//****************************************************************************************************
// Code generated by SFC Generator V1.13 on 02/04/18 16:19:18 by  MAC_IZZ from File D:\Rieckermann\old\Visio SFC\Snippet_Code\SEQ_HDR.txt
//****************************************************************************************************
//****************************************************************************************************

//================================ SEQ HEADER ================================//
//            Copyright 2018 Rieckermann Engineering Operations               //
//----------------------------------------------------------------------------//
// Title: UO_SIP_MX                                                       //
//                                                                            //
// Description:                                                               //
// Parent synchronisation flag indicating path set for filling line CIP                                                        //
//                                                                            //
// // SFC Revision History:
// Rev By               Date        CC         Note
// 0.1 Gerald Kontriner 07-Sep-2009            SFC structural design                                                       //
//----------------------------------------------------------------------------//
// Sequencer Revision History:                                                //
// Rev By               Date        CC        Note                            //
// 2.0 David Paspa      05-Jan-2018 NA        Reboot for S7-1500.             //
// 1.6 Khairul Basar    19-Nov-2009 NA        Reset #sqSequencer.STEP.Active  //
//                                            when STEP Finished.             //
// 1.5 Khairul Basar    15-Oct-2009 NA        Placeholder inserted:           //
//                                            "udtSQ_UO";          //
// 1.4 Khairul Basar    06-Oct-2009 NA        R #PAUSE;                       //
// 1.3 Khairul Basar    30-Sep-2009 NA        SEQ_HDR change STEP-0 code      //
//                                            deleted.                        //
// 1.2 Khairul Basar    26-Sep-2009 NA        Refer R4.                       //
// 1.1 Khairul Basar    23-Sep-2009 NA        Refer R3.                       //
// 1.0 Khairul Basar    20-Sep-2009 NA        STEP.Finished flag reset by     //
//                                            JUMP_MAN.                       //
// 0.9 Khairul Basar    11-Sep-2009 NA        SQ_TIMER added as VAR, declared //
//                                            in SEQ_FTR.                     //
// 0.8 Khairul Basar    09-Sep-2009 NA        SqSequencer.Err_Fault is reset  //
//                                            on Stop cmd, Step-0 dead code   //
//                                            deleted from ACT & Verify.      //
//                                            STP_FTR Step_withErr flag       //
//                                            STEP_NUM place holder           //
//                                            configured.                     //
// 0.7 Khairul Basar    28-Aug-2009 NA        SQ_FINISHED OUT added again.    //
//                                            Deleted during major mod R3.    //
// 0.6 Khairul Basar    23-Aug-2009 NA        Refer R2.                       //
// 0.5 Khairul Basar    23-Aug-2009 NA        Refer R1.                       //
// 0.4 Khairul Basar    18-Aug-2009 NA        Reset Step done with/out error  //
//                                            bits using FC:RSET.             //
// 0.3 David Paspa      16-Aug-2009 NA        Added placeholders for header   //
//                                            name and version and revision   //
//                                            history.                        //
// 0.2 Khairul Basar    11-Aug-2009 NA        Retired external udt file for   //
//                                            Static type parameters. All     //
//                                            parameters now IN, OUT or       //
//                                            IN_OUT.                         //
// 0.1 Khairul Basar    12-Jun-2009 NA        Initial design.                 //
//----------------------------------------------------------------------------//
// R4:                                                                        //
// 1.If SQ not finished Resume command will start Step timer, and redo the    //
// last action, verify the feedback.                                          //
// 2."STEP.finished" flag is ANDed with "TRN_AND_JUMP" in the snippet file    //
// TRN_HDR.This is to avoid checking of transition logic if STEP is not       //
// finished yet.                                                              //
// 3.MDCH, Load & transfer typo corrected.                                    //
//                                                                            //
// R3:                                                                        //
// 1.SqStepTimer.IN is reset in STEP_FTR instead of resetting it in TRN_HDR.  //
// This is because TRN_HDTR is not included in the Last step and StepTimer    //
// must reset in the last step.                                               //
// 2.Reset all the timers when SQ stops.Reset done in SEQ_HDR.                //
// Also STEP-finished flag reset when SQ is OFF to                            //
// scan last step.                                                            //
//                                                                            //
// R2:                                                                        //
// 1.Any step error will send the Sequencer into Pause state.Code added in    //
// SEQ_HDR.Snippet Place holder for Bool-array 8 is   //
// deleted.                                                                   //
//                                                                            //
// R1:                                                                        //
// 1.sqStepTimer:All Verification Code must satisfy the condition finish step //
// action within STEP_DELAY time(40s).If step actions not finished within the //
// time period the error flag will raise High signal.Else timer will reset.   //
// 2.sqRunTimer Added therefore can be used as retentive & non retentive.     //
// 3.sqSequencer: This is re-structured UDT which is redefined the symbol     //
// names as well as it gives more clearity.                                   //
// 4.fcMODE and fcCMD functions are added to handle the mode & command        //
// independently regardless of other logic.Two separate UDT udtMODE & udt     //
// CMD assigned to Mode & command function respectively.                      //
// 5.MAN_JUMP programed for manual mode jump operation with or without        //
// Transition code satisfied.TRN_AND_JUMP & NO_VERIFC are the parameters      //
// which will define whether verification code & transition code need to be   //
// checked to perform jump operation.                                         //
// 6.Auto to Manual switchover will be bumpless & will not affect step        //
// operation.Manual to auto switchover can be used to resume Step action at   //
// defined.                                                                   //
// Step number entered in STEPNO_JUMP.                                        //
//                                                                            //
// Parameters:                                                                //
// INPUTS                                                                     //
// ======                                                                     //
// SQ_CMD          Sequence command input inherited from object block         //
//                 0: off/idle                                                //
//                 1: start/initiate                                          //
//                 2: pause                                                   //
//                 3: resume                                                  //
//                 4: reserved (not programmed)                               //
//                 5: reserved (not programmed)                               //
//                 6: abort/go to last step                                   //
//                 7: acknowledge error/fault                                 //
// SQ_MODE         Sequencer Auto/Manual input inherited from object block    //
//                 1: manual                                                  //
//                 2: auto                                                    //
//                                                                            //
// INPUT/OUTPUTS                                                              //
// =============                                                              //
// SQ_JUMP_MAN     Allows manual jumping from one step to the next step. The  //
//                 manual jump flag is ORed with the transition process       //
//                 condition and so can be used to bypass the condition if the//
//                 sequence will not progress.                                //
//                 This input can also be used to jump to any step even       //
//                 when no transition -> step linkage exists. This is only    //
//                 possible when the SQ_MODE is in manual and SQ is in the    //
//                 idle step. The step to jump to is specified in             //
//                 SQ_man_jump_to_step (not accesseble by this FB in/out      //
//                 interface but a separate DB memory location).              //
//                                                                            //
// OUTPUTS                                                                    //
// =======                                                                    //
// SQ_STATE        The calculated state of the sequence                       //
//                 0: off/idle                                                //
//                 1: start/initiated                                         //
//                 2: paused                                                  //
//                 3: resumed                                                 //
//                 4: reserved (wrong Mode)                                   //
//                 5: reserved (Wrong commad)                                 //
//                 6: aborted/go to last step                                 //
//                 7: acknowledged error/fault                                //
// CURSTEP         Current step being proccessed.                             //
// S_ACTIVE        If current step is active                                  //
// NXT_STEP        Next step to jump to if transition condition is true       //
// ERR_FAULT       True if any error/ or fault present                        //
// PAUSED          True if step is paused                                     //
// OFF_IDLE        Sequence is not running but ready for next SQ (in step=0)  //
//----------------------------------------------------------------------------//
// Define variables:                                                          //
//----------------------------------------------------------------------------//
FUNCTION_BLOCK "fbUO_MFL_SIP_MX"
TITLE = UO : MFL_SIP_MX
NAME : FUSMX
AUTHOR : REO
VERSION : 0.1

VAR_INPUT
  MODE : INT :=2;
  SQ_CMD : INT :=0;
    _SIP_timer_complete_mx :BOOL ;	//Description
    _AUX_COND_EXn007_CMD :BOOL ;	//Description
    _TIME_DRAIN_PULSE :TIME ;	//Drain Time Setpoint
    _steam_compl_MFL_Mx :BOOL ;	//Parent synchronisation flag indicating SIP steaming is complete
    _pulse_drain_MFL_Mx :BOOL ;	//Flag indicating drain valve should be pulsed
    _ready_sip_MFL_Mx :BOOL ;	//Parent synchronisation flag for ready to start SIP
    _DEV_STATE_EXn007 :INT ;	//Device State of EXn007

END_VAR
VAR_OUTPUT
  SQ_STATE : INT ;
  CURSTEP : INT ;
  NXT_STEP : INT ;
  S_ACTIVE : BOOL ;
  ERR_FAULT : BOOL ;
  PAUSED : BOOL ;
  OFF_IDLE : BOOL ;
  SQ_FINISHED : BOOL ;
    _AUX_COND_EXn007 :BOOL ;	//Description
    _pulse_dr_compl_MFL_Mx :BOOL ;	//Pulsing of drain valve is complete
    _ready_steam_trap_MFL_Mx :BOOL ;	//Flag indicating steam traps are open
    _CMD_EXn007 :INT ;	//Command to EXn007
    _SUB_EXn007 :INT ;	//Substate selection to EXn007

END_VAR
VAR_IN_OUT
  STEPNO_JUMP : INT ;
  MAN_JUMP : BOOL ;
  NO_VERIFIC : BOOL ;
  TRN_AND_JUMP : BOOL ;

END_VAR
VAR
  sqStepTimer : "TON";
  sqRunTimer : "fbRunTimer";
  sqSequencer : "udtSQ_UO";
  SQ_TIMER: "TON";

END_VAR
BEGIN
NETWORK
TITLE =Call Mode checking function
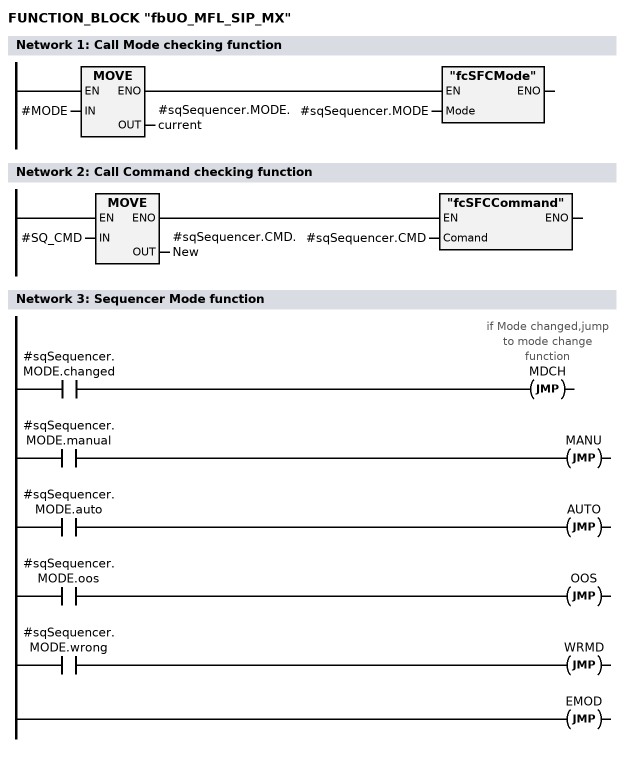

      L     #MODE;
      T     #sqSequencer.MODE.current;
      CALL "fcSFCMode" (
           Mode                     := #sqSequencer.MODE);

NETWORK
TITLE =Call Command checking function

      L     #SQ_CMD;
      T     #sqSequencer.CMD.New;

      CALL "fcSFCCommand" (
           Comand                   := #sqSequencer.CMD);

NETWORK
TITLE =Sequencer Mode function

      A     #sqSequencer.MODE.changed;
      JC    MDCH; // if Mode changed,jump to mode change function
      A     #sqSequencer.MODE.manual;
      JC    MANU;
      A     #sqSequencer.MODE.auto;
      JC    AUTO;
      A     #sqSequencer.MODE.oos;
      JC    OOS;
      A     #sqSequencer.MODE.wrong;
      JC    WRMD;
      JU    EMOD;

NETWORK
//----------------------------------------------------------------------------//
// On positive edge of mode change , this will execute once, only one cycle   //
// before going to execute the selected mode function below:                  //
//----------------------------------------------------------------------------//
TITLE =Mode change function
MDCH: NOP   0;
      SET   ;
      R     #sqStepTimer.IN;
      L     #sqSequencer.STEP.NumberCurrent;
      T     #STEPNO_JUMP;
      JU    EMOD;

NETWORK
//----------------------------------------------------------------------------//
// #TRN_AND_JUMP=can set/reset                                                //
// #sqSequencer.STEP.JumpCtrl=Can set/reset by #MAN_JUMP                      //
// #NO_VERIFIC=Can set/ Reset                                                 //
//----------------------------------------------------------------------------//
TITLE =Manual Mode function
MANU: NOP   0; //Manual mode selected



      A     #MAN_JUMP;
      =     #sqSequencer.STEP.JumpCtrl;
      A     #MAN_JUMP;
      JCN   EMOD;

      L     #STEPNO_JUMP;
      T     #sqSequencer.STEP.NumberNext;
      T     #sqSequencer.STEP.NumberCurrent;
      R     #MAN_JUMP; //Reset MAN_JUMP after loading user destination Step number
      R     #sqSequencer.STEP.Finished; //Reset finish flag, to execute next step action
      JU    EMOD;

NETWORK
//----------------------------------------------------------------------------//
// #TRN_AND_JUMP=always set                                                   //
// #sqSequencer.STEP.JumpCtrl=Always set                                      //
// #NO_VERIFIC=Alwasy Reset                                                   //
//----------------------------------------------------------------------------//
TITLE =Auto Mode function
AUTO: NOP   0; //Auto mode selected



      R     #MAN_JUMP;
      S     #TRN_AND_JUMP;
      R     #NO_VERIFIC;
      S     #sqSequencer.STEP.JumpCtrl; //Always Set in auto mode

      L     #sqSequencer.STEP.NumberCurrent;
      T     #STEPNO_JUMP;
      JU    EMOD;
NETWORK
TITLE =OOS mode function

OOS:  NOP   0; // Out of service
      JU    EMOD;
WRMD: NOP   0; //Wrong mode selected
      S     #sqSequencer.Error_Fault;
      L     "dbCONST_VAL".SQ_STATE.WRMODE;
      T     #SQ_STATE;

      JU    EMOD;

NETWORK
TITLE =Mode not changedd

      NOP   0;

NETWORK
TITLE =End Mode function

EMOD: NOP   0;

NETWORK
TITLE =An error will Pause the Sequencer,Operator must Resume SQ to run

      A     #sqSequencer.Error_Fault;
      AN    #sqSequencer.CMD.Changed;
      JC    PAUS;

NETWORK
TITLE =Command Action function

      A     #sqSequencer.CMD.Changed;
      JCN   CNCH; // if Command not changed,jump to end function
      R     #sqStepTimer.IN;


      A     #sqSequencer.CMD.Start;
      JC    STRT;

      A     #sqSequencer.CMD.Stop;
      JC    STOP;


      A     #sqSequencer.CMD.Pause;
      JC    PAUS;

      A     #sqSequencer.CMD.Resume;
      JC    RESM;

      A     #sqSequencer.CMD.Abort;
      JC    ABRT;

      A     #sqSequencer.CMD.Ack;
      JC    ACKN;

      A     #sqSequencer.CMD.wrong;
      JC    WCMD;

      JU    ECMD; //Wrong command/not specified command
//End Comand function

NETWORK
TITLE =Comand -Start/Initiate action function

STRT: NOP   0;
      R     #OFF_IDLE;
      R     #PAUSED;
      R     #sqSequencer.STEP.Active;
      R     #sqSequencer.STEP.Finished;
      R     #sqSequencer.STEP.ActionFinished;
      R     #sqSequencer.STEP.Jump;
      R     #sqSequencer.STEP.TimerExpired;
      R     #sqSequencer.STEP.Error_Fault;
      R     #sqSequencer.STEP.ActionVerified;
      R     #sqStepTimer.IN;

      S     #sqRunTimer.RESET;

//----------------------------------------------------------------------------//
// Load Initial step Number:                                                  //
//----------------------------------------------------------------------------//
      L     1;
      T     #sqSequencer.STEP.Initial;
      L     #sqSequencer.STEP.Initial;
      T     #sqSequencer.STEP.NumberCurrent;
      T     #sqSequencer.STEP.NumberNext;




      L     "dbCONST_VAL".SQ_STATE.STARTED;
      T     #SQ_STATE;

//----------------------------------------------------------------------------//
// Reset Step done without error bits:                                        //
//----------------------------------------------------------------------------//
      CALL "RSET" (
           S_BIT                    := #sqSequencer.STEP.Done[1],
           N                        := 3);//Upto final step


//----------------------------------------------------------------------------//
// Reset Step done with error bits:                                           //
//----------------------------------------------------------------------------//
      CALL "RSET" (
           S_BIT                    := #sqSequencer.STEP.WithError[1],
           N                        := 3);//Upto final step

      JU    ECMD; //End Function

NETWORK
TITLE =Comand -Stop action function

STOP: NOP   0;
      S     #OFF_IDLE;
      R     #sqSequencer.STEP.Active;
      R     #sqSequencer.STEP.Finished;
      R     #sqSequencer.STEP.ActionFinished;
      R     #sqSequencer.STEP.Jump;
      R     #sqSequencer.STEP.TimerExpired;
      R     #sqSequencer.STEP.Error_Fault;
      R     #sqSequencer.Error_Fault;
      R     #sqSequencer.STEP.ActionVerified;
      R     #sqRunTimer.ENABLE;
      R     #sqStepTimer.IN;
      R     #SQ_TIMER.IN;
      R     #PAUSED;


//Go to last step
      L     3;
      T     #sqSequencer.FinalStep;
      L     #sqSequencer.FinalStep;
      T     #sqSequencer.STEP.NumberNext;
      L     "dbCONST_VAL".SQ_STATE.OFF_IDLE;
      T     #SQ_STATE;

      JU    ECMD; //End Function

NETWORK
TITLE =Comand -Pause action function

PAUS: NOP   0;
      S     #PAUSED;
      R     #S_ACTIVE;
      S     #sqRunTimer.PAUSE;
      L     #sqSequencer.STEP.NumberCurrent;
      T     #STEPNO_JUMP;
      L     "dbCONST_VAL".SQ_STATE.PAUSED;
      T     #SQ_STATE;

      JU    ECMD; //End Function

NETWORK
TITLE =Comand -Resume action function

RESM: NOP   0;
      R     #PAUSED;
      R     #sqRunTimer.PAUSE;
      R     #sqStepTimer.IN; //Reset Step timer
      L     "dbCONST_VAL".SQ_STATE.RESUMED;
      T     #SQ_STATE;

      A     #SQ_FINISHED;
      JC    ECMD;
      R     #sqSequencer.STEP.Active;
      R     #sqSequencer.STEP.Finished;
      R     #sqSequencer.STEP.ActionFinished;

      JU    ECMD; //End Function

NETWORK
TITLE =Comand -Abort action function

ABRT: NOP   0;
      L     "dbCONST_VAL".SQ_STATE.ABORTED;
      T     #SQ_STATE;

      JC    STOP; //Stop & Abort same
      JU    ECMD;

NETWORK
TITLE =Comand -Acknowledge action function

ACKN: NOP   0;
      R     #ERR_FAULT;
      R     #sqSequencer.Error_Fault;
      L     "dbCONST_VAL".SQ_STATE.ACKNOWLEDGED;
      T     #SQ_STATE;

      JU    ECMD; //End Function

NETWORK
TITLE =Comand -wrong/unavailable

WCMD: NOP   0;

      S     #sqSequencer.Error_Fault;
      L     "dbCONST_VAL".SQ_STATE.WRCMD;
      T     #SQ_STATE;

      JU    ECMD;
NETWORK
TITLE =Comand -not changedd

CNCH: NOP   0; // Command not changed

NETWORK
TITLE =End command Function

ECMD: NOP   0;

NETWORK
//----------------------------------------------------------------------------//
// Sequencer step jump list. Load the step number to execute the step:        //
//----------------------------------------------------------------------------//
TITLE =Sequencer Step Jump distrubution list
      L     #sqSequencer.STEP.NumberCurrent;
      JL    SQER; // If Sequencer Step number invalid or greater than available number of step
      JU    S000; // Exceptional Error Handling
      JU    S001; // STEP-001:
JU    S002; // STEP-002:
JU    S003; // STEP-003:


//----------------------------------------------------------------------------//
// If Step number is Invalid or Out of Range:                                 //
//----------------------------------------------------------------------------//
SQER: NOP   0;
      S     #sqSequencer.Error_Fault;
      JU    COMM; // Jump to Common Sequencer code handling function

NETWORK
//----------------------------------------------------------------------------//
// STEP0 STEP0 STEP0 STEP0 STEP0 STEP0 STEP0 STEP0 STEP0 STEP0 STEP0 STEP0 ST //
// STEP0 STEP0 STEP0 STEP0 STEP0 STEP0 STEP0 STEP0 STEP0 STEP0 STEP0 STEP0 ST //
// STEP0 STEP0 STEP0 STEP0 STEP0 STEP0 STEP0 STEP0 STEP0 STEP0 STEP0 STEP0 ST //
//----------------------------------------------------------------------------//
TITLE =STEP0 STEP0 STEP0 STEP0 STEP0 STEP0 STEP0 STEP0 STEP0 STEP0 STEP

NETWORK
TITLE =S000: STEP0::If Paused exit

S000: NOP   0;

      JU    COMM;






NETWORK
//================================ STEP HEADER ===============================//
// STEP001 STEP001 STEP001 STEP001 ST //
// STEP001 STEP001 STEP001 STEP001 ST //
// STEP001 STEP001 STEP001 STEP001 ST //
//----------------------------------------------------------------------------//
// Set EXx014 to substate FILTER.
Set ETx003 to State DRAIN.
Open Valve DVx173.

Flag parent ready to start SIP by setting synchronization flag SIP_ready.
//----------------------------------------------------------------------------//
TITLE =S001: STEP-01::MMFLx_UO_SIP: SIP of MMFLx commenced

S001: NOP   0;

      A     #sqSequencer.CMD.Pause; //If paused jump
      JC    COMM;

NETWORK
TITLE =S001:STEP-01:Begin Action

      A     #sqSequencer.STEP.Finished;
      JC    A001; // Exit Action code, Jump to A001 Transition code

      //----------------------------------------------------------------------//
      // Begin step Action:                                                   //
      //----------------------------------------------------------------------//
      A     #sqSequencer.STEP.Active;
      JC    L001; // Action number loaded, Jump to L001--Step Action List

      //----------------------------------------------------------------------//
      // Load Default/Initial Step action number:                             //
      //----------------------------------------------------------------------//
      S     #sqSequencer.STEP.Active;
      S     #sqStepTimer.IN;
      L     1; //First Action, Step must contain Minimum one action
      T     #sqSequencer.STEP.ActionNumber;

//----------------------------------------------------------------------------//
// Step action list.                                                          //
// aann=mini Action step number(aa) inside main step number(nn)               //
// First Action aa00, Second action ab00, Third ac00, etc.                    //
//----------------------------------------------------------------------------//
L001: NOP   0;

      L     #sqSequencer.STEP.ActionNumber;
      JL    r001; //Wrong Action number
      JU    _001; //Action error handling
       JU    aa01; //ACTION-01


//----------------------------------------------------------------------------//
// More step action in the list can be inserted here, upto ab is tested:      //
//----------------------------------------------------------------------------//
r001: NOP   0; //Wrong action number
      S     #sqSequencer.Error_Fault;
      JU    k001; //Exit
_001: NOP   0; // Action error handling
      JU    k001; // Exit






NETWORK
//================================ ACT HEADER ================================//
// ACTION ACTION ACTION ACTION ACTION ACTION ACTION ACTION ACTION ACTION ACTI //
// ACTION ACTION ACTION ACTION ACTION ACTION ACTION ACTION ACTION ACTION ACTI //
// ACTION ACTION ACTION ACTION ACTION ACTION ACTION ACTION ACTION ACTION ACTI //
// ACTION ACTION ACTION ACTION ACTION ACTION ACTION ACTION ACTION ACTION ACTI //
//----------------------------------------------------------------------------//
// //Empty Step
TITLE =S001:: STEP-001:: : ACTION CODE
aa01: NOP   0;

      //----------------------------------------------------------------------//
      // ACT ACT ACT ACT ACT ACT ACT ACT ACT ACT ACT ACT ACT ACT ACT ACT ACT  //
      //----------------------------------------------------------------------//
      // Empty Step - No Action.

//----------------------------------------------------------------------------//
// VERIFY  VERIFY VERIFY VERIFY VERIFY VERIFY VERIFY VERIFY VERIFY VERIFY VER //
//----------------------------------------------------------------------------//
A M1.1; //Always High flag
      S     #sqSequencer.STEP.ActionVerified; //Action verified

      //----------------------------------------------------------------------//
      // Action done:                                                         //
      //----------------------------------------------------------------------//
      O     #sqSequencer.STEP.ActionVerified;
      O     #NO_VERIFIC; //No verification , bypass verification code
      S     #sqSequencer.STEP.ActionFinished;






      //============================= STEP FOOTER ============================//
      // Get Ready after action finished:                                     //
      //----------------------------------------------------------------------//
      A     #sqSequencer.STEP.ActionFinished;
      JCN   k001;

      //----------------------------------------------------------------------//
      // Reset Action finished flag, ready for next step action:              //
      //----------------------------------------------------------------------//
      R     #sqSequencer.STEP.ActionVerified;
      R     #sqSequencer.STEP.ActionFinished;

      //----------------------------------------------------------------------//
      // If ALL actions are finished:                                         //
      //----------------------------------------------------------------------//
      SET   ;
      S     #sqSequencer.STEP.Finished;
      R     #sqSequencer.STEP.Active;
      S     #sqSequencer.STEP.Done[01];

      //----------------------------------------------------------------------//
      // End Step action(s):                                                  //
      //----------------------------------------------------------------------//
      JU    k001;

//----------------------------------------------------------------------------//
// Finished Step Action(s):                                                   //
//----------------------------------------------------------------------------//
k001: NOP   0;

      A     #sqStepTimer.Q;
      S     #sqSequencer.STEP.WithError[01]; // Step error flag
      S     #sqSequencer.Error_Fault;
      R     #sqStepTimer.IN;
NETWORK
TITLE =S001:STEP-001::Begin Transition

A001: NOP   0;
     R     #sqStepTimer.IN;






      //============================= TRAN HEADER ============================//
      // Bypass transition if manual jump:
      //----------------------------------------------------------------------//
      A     #sqSequencer.STEP.Finished;
      A     #TRN_AND_JUMP; //Manual jump is set Transition as bypassed
      JCN   COMM; //exit

NETWORK
//----------------------------------------------------------------------------//
// TRAN   TRAN   TRAN   TRAN   TRAN   TRAN   TRAN   TRAN   TRAN   TRAN   TRAN //
// TRAN   TRAN   TRAN   TRAN   TRAN   TRAN   TRAN   TRAN   TRAN   TRAN   TRAN //
// TRAN   TRAN   TRAN   TRAN   TRAN   TRAN   TRAN   TRAN   TRAN   TRAN   TRAN //
//----------------------------------------------------------------------------//
// SIP Timer Complete
//----------------------------------------------------------------------------//
// CONDITION   CONDITION   CONDITION   CONDITION   CONDITION   CONDITION   CO //
// CONDITION   CONDITION   CONDITION   CONDITION   CONDITION   CONDITION   CO //
// CONDITION   CONDITION   CONDITION   CONDITION   CONDITION   CONDITION   CO //
//----------------------------------------------------------------------------//
TITLE =S001::STEP 001:TRAN 001: SIP Timer Complete
A #_SIP_timer_complete_mx;






      //============================= TRAN FOOTER ============================//
      // Transition jump control:                                             //
      //----------------------------------------------------------------------//
      A     #sqSequencer.STEP.JumpCtrl;
      S     #sqSequencer.STEP.Jump;

NETWORK
//----------------------------------------------------------------------------//
// Check the jump flag and jump to the next step if the transition condition  //
// is true and has set the jump flag:                                         //
//----------------------------------------------------------------------------//
TITLE =S001:t001::TRANS-v: EXIT TRANSITION AND READY THE NEXT STEP
      A     #sqSequencer.STEP.Jump;
      JCN   x001;

      R     #sqSequencer.STEP.Jump;
      R     #sqSequencer.STEP.Finished;

      L     02; // Load next STEPNO to jump to if transition satisfied
      T     #sqSequencer.STEP.NumberNext; //Next Step02.

      JU    COMM; // Transition satisfied, Exit, go to next step
x001: NOP   0;






NETWORK
//============================== STEP TRANSFER ===============================//
// Jump to the common step progression code:                                  //
//----------------------------------------------------------------------------//
TITLE =S001::STEP-001:EXIT TRANSITION:
      JU    COMM;






NETWORK
//================================ STEP HEADER ===============================//
// STEP002 STEP002 STEP002 STEP002 ST //
// STEP002 STEP002 STEP002 STEP002 ST //
// STEP002 STEP002 STEP002 STEP002 ST //
//----------------------------------------------------------------------------//
// Wait for Parent to Mx on completion drain pulse.
Wait for HPCA_blow_complete flag
Set ETx003 to State=STOPPED
//----------------------------------------------------------------------------//
TITLE =S002: STEP-02::MFL_UO_SIP_MX : Wait for complete or for drain pulse

S002: NOP   0;

      A     #sqSequencer.CMD.Pause; //If paused jump
      JC    COMM;

NETWORK
TITLE =S002:STEP-02:Begin Action

      A     #sqSequencer.STEP.Finished;
      JC    A002; // Exit Action code, Jump to A002 Transition code

      //----------------------------------------------------------------------//
      // Begin step Action:                                                   //
      //----------------------------------------------------------------------//
      A     #sqSequencer.STEP.Active;
      JC    L002; // Action number loaded, Jump to L002--Step Action List

      //----------------------------------------------------------------------//
      // Load Default/Initial Step action number:                             //
      //----------------------------------------------------------------------//
      S     #sqSequencer.STEP.Active;
      S     #sqStepTimer.IN;
      L     1; //First Action, Step must contain Minimum one action
      T     #sqSequencer.STEP.ActionNumber;

//----------------------------------------------------------------------------//
// Step action list.                                                          //
// aann=mini Action step number(aa) inside main step number(nn)               //
// First Action aa00, Second action ab00, Third ac00, etc.                    //
//----------------------------------------------------------------------------//
L002: NOP   0;

      L     #sqSequencer.STEP.ActionNumber;
      JL    r002; //Wrong Action number
      JU    _002; //Action error handling
       JU    aa02; //ACTION-01


//----------------------------------------------------------------------------//
// More step action in the list can be inserted here, upto ab is tested:      //
//----------------------------------------------------------------------------//
r002: NOP   0; //Wrong action number
      S     #sqSequencer.Error_Fault;
      JU    k002; //Exit
_002: NOP   0; // Action error handling
      JU    k002; // Exit






NETWORK
//================================ ACT HEADER ================================//
// ACTION ACTION ACTION ACTION ACTION ACTION ACTION ACTION ACTION ACTION ACTI //
// ACTION ACTION ACTION ACTION ACTION ACTION ACTION ACTION ACTION ACTION ACTI //
// ACTION ACTION ACTION ACTION ACTION ACTION ACTION ACTION ACTION ACTION ACTI //
// ACTION ACTION ACTION ACTION ACTION ACTION ACTION ACTION ACTION ACTION ACTI //
//----------------------------------------------------------------------------//
// //Set EXn007 to substate SIP_PULSE.
TITLE =S002:: STEP-002:: : ACTION CODE
aa02: NOP   0;

      //----------------------------------------------------------------------//
      // ACT ACT ACT ACT ACT ACT ACT ACT ACT ACT ACT ACT ACT ACT ACT ACT ACT  //
      //----------------------------------------------------------------------//
      L              "dbCONST_VAL".EM.EMX1.SUBS.SIP_BLK;
T 	#_SUB_EXn007;
L 	"dbCONST_VAL".EM.CMD.START;
T 	#_CMD_EXn007;
SET;
R #_pulse_dr_compl_MFL_Mx;

//----------------------------------------------------------------------------//
// VERIFY  VERIFY VERIFY VERIFY VERIFY VERIFY VERIFY VERIFY VERIFY VERIFY VER //
//----------------------------------------------------------------------------//
A(;
L #_DEV_STATE_EXn007;
L "dbCONST_VAL".EM.EMX1.SUBS.SIP_BLK;
==I;
);
      S     #sqSequencer.STEP.ActionVerified; //Action verified

      //----------------------------------------------------------------------//
      // Action done:                                                         //
      //----------------------------------------------------------------------//
      O     #sqSequencer.STEP.ActionVerified;
      O     #NO_VERIFIC; //No verification , bypass verification code
      S     #sqSequencer.STEP.ActionFinished;






      //============================= STEP FOOTER ============================//
      // Get Ready after action finished:                                     //
      //----------------------------------------------------------------------//
      A     #sqSequencer.STEP.ActionFinished;
      JCN   k002;

      //----------------------------------------------------------------------//
      // Reset Action finished flag, ready for next step action:              //
      //----------------------------------------------------------------------//
      R     #sqSequencer.STEP.ActionVerified;
      R     #sqSequencer.STEP.ActionFinished;

      //----------------------------------------------------------------------//
      // If ALL actions are finished:                                         //
      //----------------------------------------------------------------------//
      SET   ;
      S     #sqSequencer.STEP.Finished;
      R     #sqSequencer.STEP.Active;
      S     #sqSequencer.STEP.Done[02];

      //----------------------------------------------------------------------//
      // End Step action(s):                                                  //
      //----------------------------------------------------------------------//
      JU    k002;

//----------------------------------------------------------------------------//
// Finished Step Action(s):                                                   //
//----------------------------------------------------------------------------//
k002: NOP   0;

      A     #sqStepTimer.Q;
      S     #sqSequencer.STEP.WithError[02]; // Step error flag
      S     #sqSequencer.Error_Fault;
      R     #sqStepTimer.IN;
NETWORK
TITLE =S002:STEP-002::Begin Transition

A002: NOP   0;
     R     #sqStepTimer.IN;






      //============================= TRAN HEADER ============================//
      // Bypass transition if manual jump:
      //----------------------------------------------------------------------//
      A     #sqSequencer.STEP.Finished;
      A     #TRN_AND_JUMP; //Manual jump is set Transition as bypassed
      JCN   COMM; //exit

NETWORK
//----------------------------------------------------------------------------//
// TRAN   TRAN   TRAN   TRAN   TRAN   TRAN   TRAN   TRAN   TRAN   TRAN   TRAN //
// TRAN   TRAN   TRAN   TRAN   TRAN   TRAN   TRAN   TRAN   TRAN   TRAN   TRAN //
// TRAN   TRAN   TRAN   TRAN   TRAN   TRAN   TRAN   TRAN   TRAN   TRAN   TRAN //
//----------------------------------------------------------------------------//
// Wait for parent to indicate vessel steaming complete when it sets the steaming_complete flag
//----------------------------------------------------------------------------//
// CONDITION   CONDITION   CONDITION   CONDITION   CONDITION   CONDITION   CO //
// CONDITION   CONDITION   CONDITION   CONDITION   CONDITION   CONDITION   CO //
// CONDITION   CONDITION   CONDITION   CONDITION   CONDITION   CONDITION   CO //
//----------------------------------------------------------------------------//
TITLE =S002::STEP 002:TRAN 002: Vessel Steaming Complete.
A #_steam_compl_MFL_Mx;






      //============================= TRAN FOOTER ============================//
      // Transition jump control:                                             //
      //----------------------------------------------------------------------//
      A     #sqSequencer.STEP.JumpCtrl;
      S     #sqSequencer.STEP.Jump;

NETWORK
//----------------------------------------------------------------------------//
// Check the jump flag and jump to the next step if the transition condition  //
// is true and has set the jump flag:                                         //
//----------------------------------------------------------------------------//
TITLE =S002:t002::TRANS-v: EXIT TRANSITION AND READY THE NEXT STEP
      A     #sqSequencer.STEP.Jump;
      JCN   x002;

      R     #sqSequencer.STEP.Jump;
      R     #sqSequencer.STEP.Finished;

      L     03; // Load next STEPNO to jump to if transition satisfied
      T     #sqSequencer.STEP.NumberNext; //Next Step03.

      JU    COMM; // Transition satisfied, Exit, go to next step
x002: NOP   0;






NETWORK
//============================== STEP TRANSFER ===============================//
// Jump to the common step progression code:                                  //
//----------------------------------------------------------------------------//
TITLE =S002::STEP-002:EXIT TRANSITION:
      JU    COMM;






NETWORK
//================================ STEP HEADER ===============================//
// STEP003 STEP003 STEP003 STEP003 ST //
// STEP003 STEP003 STEP003 STEP003 ST //
// STEP003 STEP003 STEP003 STEP003 ST //
//----------------------------------------------------------------------------//
// Close Valve DVx173.

Set Flag MMFLx_UO_SIP completed.
//----------------------------------------------------------------------------//
TITLE =S003: STEP-03::MFL_UO_SIP: SIP of MMFLx Completed

S003: NOP   0;

      A     #sqSequencer.CMD.Pause; //If paused jump
      JC    COMM;

NETWORK
TITLE =S003:STEP-03:Begin Action

      A     #sqSequencer.STEP.Finished;
      JC    A003; // Exit Action code, Jump to A003 Transition code

      //----------------------------------------------------------------------//
      // Begin step Action:                                                   //
      //----------------------------------------------------------------------//
      A     #sqSequencer.STEP.Active;
      JC    L003; // Action number loaded, Jump to L003--Step Action List

      //----------------------------------------------------------------------//
      // Load Default/Initial Step action number:                             //
      //----------------------------------------------------------------------//
      S     #sqSequencer.STEP.Active;
      S     #sqStepTimer.IN;
      L     1; //First Action, Step must contain Minimum one action
      T     #sqSequencer.STEP.ActionNumber;

//----------------------------------------------------------------------------//
// Step action list.                                                          //
// aann=mini Action step number(aa) inside main step number(nn)               //
// First Action aa00, Second action ab00, Third ac00, etc.                    //
//----------------------------------------------------------------------------//
L003: NOP   0;

      L     #sqSequencer.STEP.ActionNumber;
      JL    r003; //Wrong Action number
      JU    _003; //Action error handling
       JU    aa03; //ACTION-01


//----------------------------------------------------------------------------//
// More step action in the list can be inserted here, upto ab is tested:      //
//----------------------------------------------------------------------------//
r003: NOP   0; //Wrong action number
      S     #sqSequencer.Error_Fault;
      JU    k003; //Exit
_003: NOP   0; // Action error handling
      JU    k003; // Exit






NETWORK
//================================ ACT HEADER ================================//
// ACTION ACTION ACTION ACTION ACTION ACTION ACTION ACTION ACTION ACTION ACTI //
// ACTION ACTION ACTION ACTION ACTION ACTION ACTION ACTION ACTION ACTION ACTI //
// ACTION ACTION ACTION ACTION ACTION ACTION ACTION ACTION ACTION ACTION ACTI //
// ACTION ACTION ACTION ACTION ACTION ACTION ACTION ACTION ACTION ACTION ACTI //
//----------------------------------------------------------------------------//
// //Set EXn007 to substate SIP_BLK.
TITLE =S003:: STEP-003:: : ACTION CODE
aa03: NOP   0;

      //----------------------------------------------------------------------//
      // ACT ACT ACT ACT ACT ACT ACT ACT ACT ACT ACT ACT ACT ACT ACT ACT ACT  //
      //----------------------------------------------------------------------//
      A             #_AUX_COND_EXn007;
JCN LEV1;
L 	"dbCONST_VAL".EM.EMX1.SUBS.SIP_BLK;
T 	#_SUB_EXn007;
L 	"dbCONST_VAL".EM.CMD.START;
T 	#_CMD_EXn007;
LEV1: NOP 0;
SET;
R #_ready_steam_trap_MFL_Mx;
R #_pulse_dr_compl_MFL_Mx;

//----------------------------------------------------------------------------//
// VERIFY  VERIFY VERIFY VERIFY VERIFY VERIFY VERIFY VERIFY VERIFY VERIFY VER //
//----------------------------------------------------------------------------//
A M1.1; //Always High flag
      S     #sqSequencer.STEP.ActionVerified; //Action verified

      //----------------------------------------------------------------------//
      // Action done:                                                         //
      //----------------------------------------------------------------------//
      O     #sqSequencer.STEP.ActionVerified;
      O     #NO_VERIFIC; //No verification , bypass verification code
      S     #sqSequencer.STEP.ActionFinished;






      //============================= STEP FOOTER ============================//
      // Get Ready after action finished:                                     //
      //----------------------------------------------------------------------//
      A     #sqSequencer.STEP.ActionFinished;
      JCN   k003;

      //----------------------------------------------------------------------//
      // Reset Action finished flag, ready for next step action:              //
      //----------------------------------------------------------------------//
      R     #sqSequencer.STEP.ActionVerified;
      R     #sqSequencer.STEP.ActionFinished;

      //----------------------------------------------------------------------//
      // If ALL actions are finished:                                         //
      //----------------------------------------------------------------------//
      SET   ;
      S     #sqSequencer.STEP.Finished;
      R     #sqSequencer.STEP.Active;
      S     #sqSequencer.STEP.Done[03];

      //----------------------------------------------------------------------//
      // End Step action(s):                                                  //
      //----------------------------------------------------------------------//
      JU    k003;

//----------------------------------------------------------------------------//
// Finished Step Action(s):                                                   //
//----------------------------------------------------------------------------//
k003: NOP   0;

      A     #sqStepTimer.Q;
      S     #sqSequencer.STEP.WithError[03]; // Step error flag
      S     #sqSequencer.Error_Fault;
      R     #sqStepTimer.IN;
NETWORK
TITLE =S003:STEP-003::Begin Transition

A003: NOP   0;
     R     #sqStepTimer.IN;






NETWORK
//============================== STEP TRANSFER ===============================//
// Jump to the common step progression code:                                  //
//----------------------------------------------------------------------------//
TITLE =S003::STEP-003:EXIT TRANSITION:
      JU    COMM;






NETWORK
//================================ SEQ FOOTER ================================//
// Common code to execute each scan:                                          //
//----------------------------------------------------------------------------//
TITLE =Sequencer Common Code, Execute in Each Scan

COMM: NOP   0;

NETWORK
TITLE =Retentive/Non Retentive Selectable Run timer

      CALL #sqRunTimer (
           TIME_H                   := #sqRunTimer.TIME_H,
           TIME_M                   := #sqRunTimer.TIME_M,
           TIME_S                   := #sqRunTimer.TIME_S,
           ENABLE                   := #sqRunTimer.ENABLE,
           RESET                    := #sqRunTimer.RESET,
           PAUSE                    := #sqRunTimer.PAUSE,
           NON_RET                  := #sqRunTimer.NON_RET,
           RMNG_H                   := #sqRunTimer.RMNG_H,
           RMNG_M                   := #sqRunTimer.RMNG_M,
           RMNG_S                   := #sqRunTimer.RMNG_S,
           TIME_EXPIRED             := #sqRunTimer.TIME_EXPIRED,
           TMR_RUNNG                := #sqRunTimer.TMR_RUNNG);

NETWORK
TITLE =Sequencer Step Timer

      CALL #sqStepTimer (
           IN                       := #sqStepTimer.IN,
           PT                       := "dbCONST_VAL".SQ_STEP_TIME,
           Q                        := #sqStepTimer.Q,
           ET                       := #sqStepTimer.ET);

NETWORK
TITLE =Sequencer Timer

 CALL #SQ_TIMER (
           IN                       := #SQ_TIMER.IN,
           PT                       := #SQ_TIMER.PT,
           Q                        := #SQ_TIMER.Q,
           ET                       := #SQ_TIMER.ET);

NETWORK
TITLE =General Assignments

      L     #sqSequencer.STEP.NumberNext;
      T     #NXT_STEP;
      T     #sqSequencer.STEP.NumberCurrent;
      T     #CURSTEP;

      A     #sqSequencer.STEP.Active;
      =     #S_ACTIVE;

      A     #sqSequencer.Error_Fault;
      =     #ERR_FAULT;

NETWORK
TITLE =Sequencer Finished

      AN    #OFF_IDLE;
      AN    #PAUSED;
      A     #sqSequencer.STEP.Done[3];
      =     #sqSequencer.Finished;
      =     #SQ_FINISHED;
      JCN   fnsd;
      L     "dbCONST_VAL".SQ_STATE.COMPLETE;
      T     #SQ_STATE;
      R     #PAUSED;
      R     #sqSequencer.STEP.Error_Fault;
      R     #sqSequencer.Error_Fault;
fnsd: NOP   0;

      //----------------------------------------------------------------------//
      // Reset Finished flag if SQ OFF for Last step to scan:                 //
      //----------------------------------------------------------------------//
      A     #OFF_IDLE;
      AN    #sqSequencer.STEP.Done[3];
      AN    #sqSequencer.STEP.WithError[3];
      JCN   abrt;
      R     #sqSequencer.STEP.Finished;
      L     "dbCONST_VAL".SQ_STATE.ABORTED;
      T     #SQ_STATE;
      S     #OFF_IDLE;
      R     #PAUSED;
      R     #sqSequencer.STEP.Error_Fault;
      R     #sqSequencer.Error_Fault;
      R     #PAUSED;
abrt: NOP   0;

//----------------------------------------------------------------------------//
// Visio Common Code Begin:                                                   //
//----------------------------------------------------------------------------//


//----------------------------------------------------------------------------//
// End of Sequencer:                                                          //
//----------------------------------------------------------------------------//
END_FUNCTION_BLOCK

